// TIA Portal V20 export
TYPE "TypeIOLinkParamData"
   STRUCT
      data { ExternalAccessible := 'False'; ExternalVisible := 'False'; ExternalWritable := 'False'} : Array[0..31] of Byte;
   END_STRUCT;
END_TYPE
